Staubli VAL3: execute.pgx

program execute(string x_sItem, bool& x_bDone[])
  local num l_nValue
  local string l_sItem
  local bool l_bOk
begin
  // compose the string
  call use:stringToArray(x_sItem,sItemsCycle)
  //
  l_bOk=true
  toNum(sItemsCycle[1],l_nValue,l_bOk)
  l_sItem=right(sItemsCycle,len(sItemsCycle)-len("OUT "))
  call out:onRun(l_sItem)
  x_bDone=true
  //
  delay(l_nValue)
  // compose the output to OFF
  l_sItem=left(l_sItem,len(l_sItem)-len(">ON"))+">OFF"
  //
  call out:onRun(l_sItem)
  x_bDone=false
end
